Fanuc KAREL source: kt00811.KL

PROGRAM KT00811
%NOLOCKGROUP
VAR
R1:REAL;R2:REAL;OUT:REAL
BEGIN
--
--
R1=2.0
R2=3.0
R1=2.0
R2=3.0
OUT=LN(R1)
END KT00811
